ABB RAPID module: Wobj_base_Nest_2.mod

MODULE Wobj_base_Nest_2
	! Points are read in order of declaration.
  ! Please do not change the order of points!

  LOCAL PERS robtarget pWobj_U_PointX1:=[[1367.143,-46.97935,-437.4996],[0.00156094937119633,0.817611932754517,0.575712502002716,0.00796413235366344],[-1,0,1,0],[9E+09,9E+09,9E+09,9E+09,9E+09,9E+09]];
	LOCAL PERS robtarget pWobj_U_PointX2:=[[1835.036,-595.9554,-438.4653],[0.0015762405237183,0.817607223987579,0.575718879699707,0.00798535905778408],[-1,0,1,0],[9E+09,9E+09,9E+09,9E+09,9E+09,9E+09]];
	LOCAL PERS robtarget pWobj_U_PointY1:=[[642.338,-661.8516,-455.5715],[0.00139784393832088,0.817752659320831,0.575513064861298,0.0079577062278986],[-1,0,0,0],[9E+09,9E+09,9E+09,9E+09,9E+09,9E+09]];

ENDMODULE
